TYPE DigitalOutput :
STRUCT
	out AT %Q*	:	BIT;
END_STRUCT
END_TYPE

(* stored: Version 1.1.0.1, ProductVersion 3.1.4020.12
   DUT DigitalOutput: Id {16246372-4cb2-4f73-908a-8fdd1dfb8155} *)
